INTERFACE I_HostMetadata EXTENDS __SYSTEM.IQueryInterface

METHOD PUBLIC AddDataAsMetadata : I_Metadata
VAR_INPUT
	Name : T_MAXSTRING;
	Data : I_Datatype;
END_VAR
END_METHOD

METHOD AddMetadata
VAR_INPUT
	Metadata : I_Metadata;
END_VAR
END_METHOD

METHOD PUBLIC TryGetMetadataByName : BOOL
VAR_INPUT
	Name : T_MAXSTRING;
	Destination : REFERENCE TO I_Metadata;
END_VAR
END_METHOD

END_INTERFACE

(* stored: Version 1.1.0.1, ProductVersion 3.1.4024.12
   Itf I_HostMetadata: Id {96f646d1-a4c9-0134-213d-25e203a1beca}
   Method AddDataAsMetadata: Id {c4dc8a5a-47d6-468e-9818-9588fa771340}
   Method AddMetadata: Id {c58c1d1e-b1d1-0e7a-041f-b8740747188f}
   Method TryGetMetadataByName: Id {8bd144a5-6123-06fd-0e73-e7fee3e3c69c} *)
